(*	HMI variables

	This block holds all HMI variables and handles communication with the HMI
	
	2024-02 HP
		-initial
*)

{attribute 'no_explicit_call' := 'do not call this POU directly'}
{attribute 'analysis' := '-33'}
FUNCTION_BLOCK HMI_LayerScan EXTENDS HMI_BaseBlock
//HMI variables that can be written to by the plc and HMI 
VAR_INPUT
	//Do not change these names, the HMI is hardcoded to use these exact names
	MAN:HMI_NotUsed;			//HMI manuals
	STS:HMI_STS_LayerScan;		//HMI statusses
	WRN:HMI_NotUsed;			//HMI warnings
	ERR:HMI_NotUsed;			//HMI errors
END_VAR

//Hmi variables that can only be written to by the HMI and read by the plc
VAR_OUTPUT PERSISTENT
	//Do not change these names, the HMI is hardcoded to use these exact names
	SP:HMI_SP_LayerScan;		//HMI setpoints
END_VAR

//this block should not be called

END_FUNCTION_BLOCK

(* stored: Version 1.1.0.1
   POU HMI_LayerScan: Id {fd98de95-229e-4f1a-8ab2-c53cb39054a7}, SpecialFunc None *)
